// TIA Portal V17 export
// export: Created 2023-10-17T06:55:20.9500846Z, ExportSetting WithDefaults, DisplayName Totally Integrated Automation Portal, DisplayVersion V17, DisplayName TIA Portal Openness, DisplayVersion V17, DisplayName TIA Portal Version Control Interface, DisplayVersion V17, DisplayName STEP 7 Professional, DisplayVersion V17, DisplayName STEP 7 Safety, DisplayVersion V17, DisplayName WinCC Advanced, DisplayVersion V17
DATA_BLOCK "Device"   // DB1
{ S7_Optimized_Access := 'FALSE' }
VERSION : 0.1
// stored: AutoNumber true, DBAccessibleFromOPCUA true, DBAccessibleFromWebserver true, IsOnlyStoredInLoadMemory false, IsWriteProtectedInAS false
   VAR
      V1103 : Bool;
      V01101 : Bool;
      V2101 : Bool;
      V3101 : Bool;
      V1102 : Bool;
      V2102 : Bool;
      V3102 : Bool;
      V4101 : Bool;
      V4102 : Bool;
      V4103 : Bool;
      W1111 : Real;
      W2111 : Real;
      W3111 : Real;
      L4141 : Real;
      AGR5101 : Bool;
      PUMP4121 : Bool;
      PASTEURISING_MACHINE_ON : Bool;
      FILLING_MACHINE : Bool;
      V1101 : Bool;
      L5141 : Real;
      V01101_s : Bool;
      V2101_s : Bool;
      V3101_s : Bool;
      V1102_s : Bool;
      V2102_s : Bool;
      V3102_s : Bool;
      AGR5101_s : Bool;
      V4101_s : Bool;
      PUMP4121_s : Bool;
      V4102_s : Bool;
      PASTEURISING_MACHINE_ON_s : Bool;
      FILLING_MACHINE_s : Bool;
      V2102_ss : Bool;
      V4103_s : Bool;
   END_VAR
BEGIN
END_DATA_BLOCK
